BEGIN
   Zulauf_AR_Niv.EW_Peri := 16#287C;
   Zulauf_AR_Niv.EW_PW := 0.0;
   Zulauf_AR_Niv.E.St := FALSE;
   Zulauf_AR_Niv.E.Wt := FALSE;
   Zulauf_AR_Niv.E.Kom_DP := FALSE;
   Zulauf_AR_Niv.E.Kom_int := FALSE;
   Zulauf_AR_Niv.E.int_St := FALSE;
   Zulauf_AR_Niv.E.MW_OF_St := FALSE;
   Zulauf_AR_Niv.E.MW_inv_St := FALSE;
   Zulauf_AR_Niv.E.ZI := FALSE;
   Zulauf_AR_Niv.E.AF_St := FALSE;
   Zulauf_AR_Niv.E.Res09 := FALSE;
   Zulauf_AR_Niv.E.Res10 := FALSE;
   Zulauf_AR_Niv.E.Res11 := FALSE;
   Zulauf_AR_Niv.E.Res12 := FALSE;
   Zulauf_AR_Niv.E.Res13 := FALSE;
   Zulauf_AR_Niv.E.Res14 := FALSE;
   Zulauf_AR_Niv.E.Res15 := FALSE;
   Zulauf_AR_Temp.EW_Peri := 16#1599;
   Zulauf_AR_Temp.EW_PW := 0.0;
   Zulauf_AR_Temp.E.St := FALSE;
   Zulauf_AR_Temp.E.Wt := FALSE;
   Zulauf_AR_Temp.E.Kom_DP := FALSE;
   Zulauf_AR_Temp.E.Kom_int := FALSE;
   Zulauf_AR_Temp.E.int_St := FALSE;
   Zulauf_AR_Temp.E.MW_OF_St := FALSE;
   Zulauf_AR_Temp.E.MW_inv_St := FALSE;
   Zulauf_AR_Temp.E.ZI := FALSE;
   Zulauf_AR_Temp.E.AF_St := FALSE;
   Zulauf_AR_Temp.E.Res09 := FALSE;
   Zulauf_AR_Temp.E.Res10 := FALSE;
   Zulauf_AR_Temp.E.Res11 := FALSE;
   Zulauf_AR_Temp.E.Res12 := FALSE;
   Zulauf_AR_Temp.E.Res13 := FALSE;
   Zulauf_AR_Temp.E.Res14 := FALSE;
   Zulauf_AR_Temp.E.Res15 := FALSE;
   Zulauf_AR_DF.EW_Peri := 16#0000;
   Zulauf_AR_DF.EW_PW := 0.0;
   Zulauf_AR_DF.E.St := FALSE;
   Zulauf_AR_DF.E.Wt := FALSE;
   Zulauf_AR_DF.E.Kom_DP := FALSE;
   Zulauf_AR_DF.E.Kom_int := FALSE;
   Zulauf_AR_DF.E.int_St := FALSE;
   Zulauf_AR_DF.E.MW_OF_St := FALSE;
   Zulauf_AR_DF.E.MW_inv_St := FALSE;
   Zulauf_AR_DF.E.ZI := FALSE;
   Zulauf_AR_DF.E.AF_St := FALSE;
   Zulauf_AR_DF.E.Res09 := FALSE;
   Zulauf_AR_DF.E.Res10 := FALSE;
   Zulauf_AR_DF.E.Res11 := FALSE;
   Zulauf_AR_DF.E.Res12 := FALSE;
   Zulauf_AR_DF.E.Res13 := FALSE;
   Zulauf_AR_DF.E.Res14 := FALSE;
   Zulauf_AR_DF.E.Res15 := FALSE;
   BB1_AS1_SS.EW_Peri := 16#1599;
   BB1_AS1_SS.EW_PW := 0.0;
   BB1_AS1_SS.E.St := FALSE;
   BB1_AS1_SS.E.Wt := FALSE;
   BB1_AS1_SS.E.Kom_DP := FALSE;
   BB1_AS1_SS.E.Kom_int := FALSE;
   BB1_AS1_SS.E.int_St := FALSE;
   BB1_AS1_SS.E.MW_OF_St := FALSE;
   BB1_AS1_SS.E.MW_inv_St := FALSE;
   BB1_AS1_SS.E.ZI := FALSE;
   BB1_AS1_SS.E.AF_St := FALSE;
   BB1_AS1_SS.E.Res09 := FALSE;
   BB1_AS1_SS.E.Res10 := FALSE;
   BB1_AS1_SS.E.Res11 := FALSE;
   BB1_AS1_SS.E.Res12 := FALSE;
   BB1_AS1_SS.E.Res13 := FALSE;
   BB1_AS1_SS.E.Res14 := FALSE;
   BB1_AS1_SS.E.Res15 := FALSE;
   BB1_AS2_SS.EW_Peri := 16#57CD;
   BB1_AS2_SS.EW_PW := 0.0;
   BB1_AS2_SS.E.St := FALSE;
   BB1_AS2_SS.E.Wt := FALSE;
   BB1_AS2_SS.E.Kom_DP := FALSE;
   BB1_AS2_SS.E.Kom_int := FALSE;
   BB1_AS2_SS.E.int_St := FALSE;
   BB1_AS2_SS.E.MW_OF_St := FALSE;
   BB1_AS2_SS.E.MW_inv_St := FALSE;
   BB1_AS2_SS.E.ZI := FALSE;
   BB1_AS2_SS.E.AF_St := FALSE;
   BB1_AS2_SS.E.Res09 := FALSE;
   BB1_AS2_SS.E.Res10 := FALSE;
   BB1_AS2_SS.E.Res11 := FALSE;
   BB1_AS2_SS.E.Res12 := FALSE;
   BB1_AS2_SS.E.Res13 := FALSE;
   BB1_AS2_SS.E.Res14 := FALSE;
   BB1_AS2_SS.E.Res15 := FALSE;
   BB2_AS1_SS.EW_Peri := 16#15A5;
   BB2_AS1_SS.EW_PW := 0.0;
   BB2_AS1_SS.E.St := FALSE;
   BB2_AS1_SS.E.Wt := FALSE;
   BB2_AS1_SS.E.Kom_DP := FALSE;
   BB2_AS1_SS.E.Kom_int := FALSE;
   BB2_AS1_SS.E.int_St := FALSE;
   BB2_AS1_SS.E.MW_OF_St := FALSE;
   BB2_AS1_SS.E.MW_inv_St := FALSE;
   BB2_AS1_SS.E.ZI := FALSE;
   BB2_AS1_SS.E.AF_St := FALSE;
   BB2_AS1_SS.E.Res09 := FALSE;
   BB2_AS1_SS.E.Res10 := FALSE;
   BB2_AS1_SS.E.Res11 := FALSE;
   BB2_AS1_SS.E.Res12 := FALSE;
   BB2_AS1_SS.E.Res13 := FALSE;
   BB2_AS1_SS.E.Res14 := FALSE;
   BB2_AS1_SS.E.Res15 := FALSE;
   BB2_AS2_SS.EW_Peri := 16#15B8;
   BB2_AS2_SS.EW_PW := 0.0;
   BB2_AS2_SS.E.St := FALSE;
   BB2_AS2_SS.E.Wt := FALSE;
   BB2_AS2_SS.E.Kom_DP := FALSE;
   BB2_AS2_SS.E.Kom_int := FALSE;
   BB2_AS2_SS.E.int_St := FALSE;
   BB2_AS2_SS.E.MW_OF_St := FALSE;
   BB2_AS2_SS.E.MW_inv_St := FALSE;
   BB2_AS2_SS.E.ZI := FALSE;
   BB2_AS2_SS.E.AF_St := FALSE;
   BB2_AS2_SS.E.Res09 := FALSE;
   BB2_AS2_SS.E.Res10 := FALSE;
   BB2_AS2_SS.E.Res11 := FALSE;
   BB2_AS2_SS.E.Res12 := FALSE;
   BB2_AS2_SS.E.Res13 := FALSE;
   BB2_AS2_SS.E.Res14 := FALSE;
   BB2_AS2_SS.E.Res15 := FALSE;
   BB1_O2.EW_Peri := 16#235C;
   BB1_O2.EW_PW := 0.0;
   BB1_O2.E.St := FALSE;
   BB1_O2.E.Wt := FALSE;
   BB1_O2.E.Kom_DP := FALSE;
   BB1_O2.E.Kom_int := FALSE;
   BB1_O2.E.int_St := FALSE;
   BB1_O2.E.MW_OF_St := FALSE;
   BB1_O2.E.MW_inv_St := FALSE;
   BB1_O2.E.ZI := FALSE;
   BB1_O2.E.AF_St := FALSE;
   BB1_O2.E.Res09 := FALSE;
   BB1_O2.E.Res10 := FALSE;
   BB1_O2.E.Res11 := FALSE;
   BB1_O2.E.Res12 := FALSE;
   BB1_O2.E.Res13 := FALSE;
   BB1_O2.E.Res14 := FALSE;
   BB1_O2.E.Res15 := FALSE;
   BB1_Temp.EW_Peri := 16#2EBA;
   BB1_Temp.EW_PW := 0.0;
   BB1_Temp.E.St := FALSE;
   BB1_Temp.E.Wt := FALSE;
   BB1_Temp.E.Kom_DP := FALSE;
   BB1_Temp.E.Kom_int := FALSE;
   BB1_Temp.E.int_St := FALSE;
   BB1_Temp.E.MW_OF_St := FALSE;
   BB1_Temp.E.MW_inv_St := FALSE;
   BB1_Temp.E.ZI := FALSE;
   BB1_Temp.E.AF_St := FALSE;
   BB1_Temp.E.Res09 := FALSE;
   BB1_Temp.E.Res10 := FALSE;
   BB1_Temp.E.Res11 := FALSE;
   BB1_Temp.E.Res12 := FALSE;
   BB1_Temp.E.Res13 := FALSE;
   BB1_Temp.E.Res14 := FALSE;
   BB1_Temp.E.Res15 := FALSE;
   BB2_O2.EW_Peri := 16#2288;
   BB2_O2.EW_PW := 0.0;
   BB2_O2.E.St := FALSE;
   BB2_O2.E.Wt := FALSE;
   BB2_O2.E.Kom_DP := FALSE;
   BB2_O2.E.Kom_int := FALSE;
   BB2_O2.E.int_St := FALSE;
   BB2_O2.E.MW_OF_St := FALSE;
   BB2_O2.E.MW_inv_St := FALSE;
   BB2_O2.E.ZI := FALSE;
   BB2_O2.E.AF_St := FALSE;
   BB2_O2.E.Res09 := FALSE;
   BB2_O2.E.Res10 := FALSE;
   BB2_O2.E.Res11 := FALSE;
   BB2_O2.E.Res12 := FALSE;
   BB2_O2.E.Res13 := FALSE;
   BB2_O2.E.Res14 := FALSE;
   BB2_O2.E.Res15 := FALSE;
   BB2_Temp.EW_Peri := 16#2E74;
   BB2_Temp.EW_PW := 0.0;
   BB2_Temp.E.St := FALSE;
   BB2_Temp.E.Wt := FALSE;
   BB2_Temp.E.Kom_DP := FALSE;
   BB2_Temp.E.Kom_int := FALSE;
   BB2_Temp.E.int_St := FALSE;
   BB2_Temp.E.MW_OF_St := FALSE;
   BB2_Temp.E.MW_inv_St := FALSE;
   BB2_Temp.E.ZI := FALSE;
   BB2_Temp.E.AF_St := FALSE;
   BB2_Temp.E.Res09 := FALSE;
   BB2_Temp.E.Res10 := FALSE;
   BB2_Temp.E.Res11 := FALSE;
   BB2_Temp.E.Res12 := FALSE;
   BB2_Temp.E.Res13 := FALSE;
   BB2_Temp.E.Res14 := FALSE;
   BB2_Temp.E.Res15 := FALSE;
   BB1_DF.EW_Peri := 16#1599;
   BB1_DF.EW_PW := 0.0;
   BB1_DF.E.St := FALSE;
   BB1_DF.E.Wt := FALSE;
   BB1_DF.E.Kom_DP := FALSE;
   BB1_DF.E.Kom_int := FALSE;
   BB1_DF.E.int_St := FALSE;
   BB1_DF.E.MW_OF_St := FALSE;
   BB1_DF.E.MW_inv_St := FALSE;
   BB1_DF.E.ZI := FALSE;
   BB1_DF.E.AF_St := FALSE;
   BB1_DF.E.Res09 := FALSE;
   BB1_DF.E.Res10 := FALSE;
   BB1_DF.E.Res11 := FALSE;
   BB1_DF.E.Res12 := FALSE;
   BB1_DF.E.Res13 := FALSE;
   BB1_DF.E.Res14 := FALSE;
   BB1_DF.E.Res15 := FALSE;
   BB2_DF.EW_Peri := 16#1599;
   BB2_DF.EW_PW := 0.0;
   BB2_DF.E.St := FALSE;
   BB2_DF.E.Wt := FALSE;
   BB2_DF.E.Kom_DP := FALSE;
   BB2_DF.E.Kom_int := FALSE;
   BB2_DF.E.int_St := FALSE;
   BB2_DF.E.MW_OF_St := FALSE;
   BB2_DF.E.MW_inv_St := FALSE;
   BB2_DF.E.ZI := FALSE;
   BB2_DF.E.AF_St := FALSE;
   BB2_DF.E.Res09 := FALSE;
   BB2_DF.E.Res10 := FALSE;
   BB2_DF.E.Res11 := FALSE;
   BB2_DF.E.Res12 := FALSE;
   BB2_DF.E.Res13 := FALSE;
   BB2_DF.E.Res14 := FALSE;
   BB2_DF.E.Res15 := FALSE;
   Zulauf_Niv.EW_Peri := 16#2C3F;
   Zulauf_Niv.EW_PW := 0.0;
   Zulauf_Niv.E.St := FALSE;
   Zulauf_Niv.E.Wt := FALSE;
   Zulauf_Niv.E.Kom_DP := FALSE;
   Zulauf_Niv.E.Kom_int := FALSE;
   Zulauf_Niv.E.int_St := FALSE;
   Zulauf_Niv.E.MW_OF_St := FALSE;
   Zulauf_Niv.E.MW_inv_St := FALSE;
   Zulauf_Niv.E.ZI := FALSE;
   Zulauf_Niv.E.AF_St := FALSE;
   Zulauf_Niv.E.Res09 := FALSE;
   Zulauf_Niv.E.Res10 := FALSE;
   Zulauf_Niv.E.Res11 := FALSE;
   Zulauf_Niv.E.Res12 := FALSE;
   Zulauf_Niv.E.Res13 := FALSE;
   Zulauf_Niv.E.Res14 := FALSE;
   Zulauf_Niv.E.Res15 := FALSE;
   Zulauf_DF.EW_Peri := 16#39D4;
   Zulauf_DF.EW_PW := 0.0;
   Zulauf_DF.E.St := FALSE;
   Zulauf_DF.E.Wt := FALSE;
   Zulauf_DF.E.Kom_DP := FALSE;
   Zulauf_DF.E.Kom_int := FALSE;
   Zulauf_DF.E.int_St := FALSE;
   Zulauf_DF.E.MW_OF_St := FALSE;
   Zulauf_DF.E.MW_inv_St := FALSE;
   Zulauf_DF.E.ZI := FALSE;
   Zulauf_DF.E.AF_St := FALSE;
   Zulauf_DF.E.Res09 := FALSE;
   Zulauf_DF.E.Res10 := FALSE;
   Zulauf_DF.E.Res11 := FALSE;
   Zulauf_DF.E.Res12 := FALSE;
   Zulauf_DF.E.Res13 := FALSE;
   Zulauf_DF.E.Res14 := FALSE;
   Zulauf_DF.E.Res15 := FALSE;
   Verteiler_pH.EW_Peri := 16#1599;
   Verteiler_pH.EW_PW := 0.0;
   Verteiler_pH.E.St := FALSE;
   Verteiler_pH.E.Wt := FALSE;
   Verteiler_pH.E.Kom_DP := FALSE;
   Verteiler_pH.E.Kom_int := FALSE;
   Verteiler_pH.E.int_St := FALSE;
   Verteiler_pH.E.MW_OF_St := FALSE;
   Verteiler_pH.E.MW_inv_St := FALSE;
   Verteiler_pH.E.ZI := FALSE;
   Verteiler_pH.E.AF_St := FALSE;
   Verteiler_pH.E.Res09 := FALSE;
   Verteiler_pH.E.Res10 := FALSE;
   Verteiler_pH.E.Res11 := FALSE;
   Verteiler_pH.E.Res12 := FALSE;
   Verteiler_pH.E.Res13 := FALSE;
   Verteiler_pH.E.Res14 := FALSE;
   Verteiler_pH.E.Res15 := FALSE;
   Verteiler_O2.EW_Peri := 16#1599;
   Verteiler_O2.EW_PW := 0.0;
   Verteiler_O2.E.St := FALSE;
   Verteiler_O2.E.Wt := FALSE;
   Verteiler_O2.E.Kom_DP := FALSE;
   Verteiler_O2.E.Kom_int := FALSE;
   Verteiler_O2.E.int_St := FALSE;
   Verteiler_O2.E.MW_OF_St := FALSE;
   Verteiler_O2.E.MW_inv_St := FALSE;
   Verteiler_O2.E.ZI := FALSE;
   Verteiler_O2.E.AF_St := FALSE;
   Verteiler_O2.E.Res09 := FALSE;
   Verteiler_O2.E.Res10 := FALSE;
   Verteiler_O2.E.Res11 := FALSE;
   Verteiler_O2.E.Res12 := FALSE;
   Verteiler_O2.E.Res13 := FALSE;
   Verteiler_O2.E.Res14 := FALSE;
   Verteiler_O2.E.Res15 := FALSE;
   Verteiler_Temp.EW_Peri := 16#1599;
   Verteiler_Temp.EW_PW := 0.0;
   Verteiler_Temp.E.St := FALSE;
   Verteiler_Temp.E.Wt := FALSE;
   Verteiler_Temp.E.Kom_DP := FALSE;
   Verteiler_Temp.E.Kom_int := FALSE;
   Verteiler_Temp.E.int_St := FALSE;
   Verteiler_Temp.E.MW_OF_St := FALSE;
   Verteiler_Temp.E.MW_inv_St := FALSE;
   Verteiler_Temp.E.ZI := FALSE;
   Verteiler_Temp.E.AF_St := FALSE;
   Verteiler_Temp.E.Res09 := FALSE;
   Verteiler_Temp.E.Res10 := FALSE;
   Verteiler_Temp.E.Res11 := FALSE;
   Verteiler_Temp.E.Res12 := FALSE;
   Verteiler_Temp.E.Res13 := FALSE;
   Verteiler_Temp.E.Res14 := FALSE;
   Verteiler_Temp.E.Res15 := FALSE;
   BB_UeSS_DF.EW_Peri := 16#1592;
   BB_UeSS_DF.EW_PW := 0.0;
   BB_UeSS_DF.E.St := FALSE;
   BB_UeSS_DF.E.Wt := FALSE;
   BB_UeSS_DF.E.Kom_DP := FALSE;
   BB_UeSS_DF.E.Kom_int := FALSE;
   BB_UeSS_DF.E.int_St := FALSE;
   BB_UeSS_DF.E.MW_OF_St := FALSE;
   BB_UeSS_DF.E.MW_inv_St := FALSE;
   BB_UeSS_DF.E.ZI := FALSE;
   BB_UeSS_DF.E.AF_St := FALSE;
   BB_UeSS_DF.E.Res09 := FALSE;
   BB_UeSS_DF.E.Res10 := FALSE;
   BB_UeSS_DF.E.Res11 := FALSE;
   BB_UeSS_DF.E.Res12 := FALSE;
   BB_UeSS_DF.E.Res13 := FALSE;
   BB_UeSS_DF.E.Res14 := FALSE;
   BB_UeSS_DF.E.Res15 := FALSE;
   Ablauf_DF.EW_Peri := 16#35E9;
   Ablauf_DF.EW_PW := 0.0;
   Ablauf_DF.E.St := FALSE;
   Ablauf_DF.E.Wt := FALSE;
   Ablauf_DF.E.Kom_DP := FALSE;
   Ablauf_DF.E.Kom_int := FALSE;
   Ablauf_DF.E.int_St := FALSE;
   Ablauf_DF.E.MW_OF_St := FALSE;
   Ablauf_DF.E.MW_inv_St := FALSE;
   Ablauf_DF.E.ZI := FALSE;
   Ablauf_DF.E.AF_St := FALSE;
   Ablauf_DF.E.Res09 := FALSE;
   Ablauf_DF.E.Res10 := FALSE;
   Ablauf_DF.E.Res11 := FALSE;
   Ablauf_DF.E.Res12 := FALSE;
   Ablauf_DF.E.Res13 := FALSE;
   Ablauf_DF.E.Res14 := FALSE;
   Ablauf_DF.E.Res15 := FALSE;
   Ablauf_pH.EW_Peri := 16#4122;
   Ablauf_pH.EW_PW := 0.0;
   Ablauf_pH.E.St := FALSE;
   Ablauf_pH.E.Wt := FALSE;
   Ablauf_pH.E.Kom_DP := FALSE;
   Ablauf_pH.E.Kom_int := FALSE;
   Ablauf_pH.E.int_St := FALSE;
   Ablauf_pH.E.MW_OF_St := FALSE;
   Ablauf_pH.E.MW_inv_St := FALSE;
   Ablauf_pH.E.ZI := FALSE;
   Ablauf_pH.E.AF_St := FALSE;
   Ablauf_pH.E.Res09 := FALSE;
   Ablauf_pH.E.Res10 := FALSE;
   Ablauf_pH.E.Res11 := FALSE;
   Ablauf_pH.E.Res12 := FALSE;
   Ablauf_pH.E.Res13 := FALSE;
   Ablauf_pH.E.Res14 := FALSE;
   Ablauf_pH.E.Res15 := FALSE;
   Ablauf_O2.EW_Peri := 16#225E;
   Ablauf_O2.EW_PW := 0.0;
   Ablauf_O2.E.St := FALSE;
   Ablauf_O2.E.Wt := FALSE;
   Ablauf_O2.E.Kom_DP := FALSE;
   Ablauf_O2.E.Kom_int := FALSE;
   Ablauf_O2.E.int_St := FALSE;
   Ablauf_O2.E.MW_OF_St := FALSE;
   Ablauf_O2.E.MW_inv_St := FALSE;
   Ablauf_O2.E.ZI := FALSE;
   Ablauf_O2.E.AF_St := FALSE;
   Ablauf_O2.E.Res09 := FALSE;
   Ablauf_O2.E.Res10 := FALSE;
   Ablauf_O2.E.Res11 := FALSE;
   Ablauf_O2.E.Res12 := FALSE;
   Ablauf_O2.E.Res13 := FALSE;
   Ablauf_O2.E.Res14 := FALSE;
   Ablauf_O2.E.Res15 := FALSE;
   Ablauf_Temp.EW_Peri := 16#2BEC;
   Ablauf_Temp.EW_PW := 0.0;
   Ablauf_Temp.E.St := FALSE;
   Ablauf_Temp.E.Wt := FALSE;
   Ablauf_Temp.E.Kom_DP := FALSE;
   Ablauf_Temp.E.Kom_int := FALSE;
   Ablauf_Temp.E.int_St := FALSE;
   Ablauf_Temp.E.MW_OF_St := FALSE;
   Ablauf_Temp.E.MW_inv_St := FALSE;
   Ablauf_Temp.E.ZI := FALSE;
   Ablauf_Temp.E.AF_St := FALSE;
   Ablauf_Temp.E.Res09 := FALSE;
   Ablauf_Temp.E.Res10 := FALSE;
   Ablauf_Temp.E.Res11 := FALSE;
   Ablauf_Temp.E.Res12 := FALSE;
   Ablauf_Temp.E.Res13 := FALSE;
   Ablauf_Temp.E.Res14 := FALSE;
   Ablauf_Temp.E.Res15 := FALSE;
   Schlamm_ED_Niv.EW_Peri := 16#1599;
   Schlamm_ED_Niv.EW_PW := 0.0;
   Schlamm_ED_Niv.E.St := FALSE;
   Schlamm_ED_Niv.E.Wt := FALSE;
   Schlamm_ED_Niv.E.Kom_DP := FALSE;
   Schlamm_ED_Niv.E.Kom_int := FALSE;
   Schlamm_ED_Niv.E.int_St := FALSE;
   Schlamm_ED_Niv.E.MW_OF_St := FALSE;
   Schlamm_ED_Niv.E.MW_inv_St := FALSE;
   Schlamm_ED_Niv.E.ZI := FALSE;
   Schlamm_ED_Niv.E.AF_St := FALSE;
   Schlamm_ED_Niv.E.Res09 := FALSE;
   Schlamm_ED_Niv.E.Res10 := FALSE;
   Schlamm_ED_Niv.E.Res11 := FALSE;
   Schlamm_ED_Niv.E.Res12 := FALSE;
   Schlamm_ED_Niv.E.Res13 := FALSE;
   Schlamm_ED_Niv.E.Res14 := FALSE;
   Schlamm_ED_Niv.E.Res15 := FALSE;
   Schlamm_Besch_Niv.EW_Peri := 16#1599;
   Schlamm_Besch_Niv.EW_PW := 0.0;
   Schlamm_Besch_Niv.E.St := FALSE;
   Schlamm_Besch_Niv.E.Wt := FALSE;
   Schlamm_Besch_Niv.E.Kom_DP := FALSE;
   Schlamm_Besch_Niv.E.Kom_int := FALSE;
   Schlamm_Besch_Niv.E.int_St := FALSE;
   Schlamm_Besch_Niv.E.MW_OF_St := FALSE;
   Schlamm_Besch_Niv.E.MW_inv_St := FALSE;
   Schlamm_Besch_Niv.E.ZI := FALSE;
   Schlamm_Besch_Niv.E.AF_St := FALSE;
   Schlamm_Besch_Niv.E.Res09 := FALSE;
   Schlamm_Besch_Niv.E.Res10 := FALSE;
   Schlamm_Besch_Niv.E.Res11 := FALSE;
   Schlamm_Besch_Niv.E.Res12 := FALSE;
   Schlamm_Besch_Niv.E.Res13 := FALSE;
   Schlamm_Besch_Niv.E.Res14 := FALSE;
   Schlamm_Besch_Niv.E.Res15 := FALSE;
   Schlamm_Besch_DF.EW_Peri := 16#159B;
   Schlamm_Besch_DF.EW_PW := 0.0;
   Schlamm_Besch_DF.E.St := FALSE;
   Schlamm_Besch_DF.E.Wt := FALSE;
   Schlamm_Besch_DF.E.Kom_DP := FALSE;
   Schlamm_Besch_DF.E.Kom_int := FALSE;
   Schlamm_Besch_DF.E.int_St := FALSE;
   Schlamm_Besch_DF.E.MW_OF_St := FALSE;
   Schlamm_Besch_DF.E.MW_inv_St := FALSE;
   Schlamm_Besch_DF.E.ZI := FALSE;
   Schlamm_Besch_DF.E.AF_St := FALSE;
   Schlamm_Besch_DF.E.Res09 := FALSE;
   Schlamm_Besch_DF.E.Res10 := FALSE;
   Schlamm_Besch_DF.E.Res11 := FALSE;
   Schlamm_Besch_DF.E.Res12 := FALSE;
   Schlamm_Besch_DF.E.Res13 := FALSE;
   Schlamm_Besch_DF.E.Res14 := FALSE;
   Schlamm_Besch_DF.E.Res15 := FALSE;
   Truebwasser_Niv.EW_Peri := 16#28E3;
   Truebwasser_Niv.EW_PW := 0.0;
   Truebwasser_Niv.E.St := FALSE;
   Truebwasser_Niv.E.Wt := FALSE;
   Truebwasser_Niv.E.Kom_DP := FALSE;
   Truebwasser_Niv.E.Kom_int := FALSE;
   Truebwasser_Niv.E.int_St := FALSE;
   Truebwasser_Niv.E.MW_OF_St := FALSE;
   Truebwasser_Niv.E.MW_inv_St := FALSE;
   Truebwasser_Niv.E.ZI := FALSE;
   Truebwasser_Niv.E.AF_St := FALSE;
   Truebwasser_Niv.E.Res09 := FALSE;
   Truebwasser_Niv.E.Res10 := FALSE;
   Truebwasser_Niv.E.Res11 := FALSE;
   Truebwasser_Niv.E.Res12 := FALSE;
   Truebwasser_Niv.E.Res13 := FALSE;
   Truebwasser_Niv.E.Res14 := FALSE;
   Truebwasser_Niv.E.Res15 := FALSE;
   Truebwasser_DF.EW_Peri := 16#1597;
   Truebwasser_DF.EW_PW := 0.0;
   Truebwasser_DF.E.St := FALSE;
   Truebwasser_DF.E.Wt := FALSE;
   Truebwasser_DF.E.Kom_DP := FALSE;
   Truebwasser_DF.E.Kom_int := FALSE;
   Truebwasser_DF.E.int_St := FALSE;
   Truebwasser_DF.E.MW_OF_St := FALSE;
   Truebwasser_DF.E.MW_inv_St := FALSE;
   Truebwasser_DF.E.ZI := FALSE;
   Truebwasser_DF.E.AF_St := FALSE;
   Truebwasser_DF.E.Res09 := FALSE;
   Truebwasser_DF.E.Res10 := FALSE;
   Truebwasser_DF.E.Res11 := FALSE;
   Truebwasser_DF.E.Res12 := FALSE;
   Truebwasser_DF.E.Res13 := FALSE;
   Truebwasser_DF.E.Res14 := FALSE;
   Truebwasser_DF.E.Res15 := FALSE;
   Zulauf_SF_Niv.EW_Peri := 16#1599;
   Zulauf_SF_Niv.EW_PW := 0.0;
   Zulauf_SF_Niv.E.St := FALSE;
   Zulauf_SF_Niv.E.Wt := FALSE;
   Zulauf_SF_Niv.E.Kom_DP := FALSE;
   Zulauf_SF_Niv.E.Kom_int := FALSE;
   Zulauf_SF_Niv.E.int_St := FALSE;
   Zulauf_SF_Niv.E.MW_OF_St := FALSE;
   Zulauf_SF_Niv.E.MW_inv_St := FALSE;
   Zulauf_SF_Niv.E.ZI := FALSE;
   Zulauf_SF_Niv.E.AF_St := FALSE;
   Zulauf_SF_Niv.E.Res09 := FALSE;
   Zulauf_SF_Niv.E.Res10 := FALSE;
   Zulauf_SF_Niv.E.Res11 := FALSE;
   Zulauf_SF_Niv.E.Res12 := FALSE;
   Zulauf_SF_Niv.E.Res13 := FALSE;
   Zulauf_SF_Niv.E.Res14 := FALSE;
   Zulauf_SF_Niv.E.Res15 := FALSE;
   Ablauf_NOx.EW_Peri := 16#1BEB;
   Ablauf_NOx.EW_PW := 0.0;
   Ablauf_NOx.E.St := FALSE;
   Ablauf_NOx.E.Wt := FALSE;
   Ablauf_NOx.E.Kom_DP := FALSE;
   Ablauf_NOx.E.Kom_int := FALSE;
   Ablauf_NOx.E.int_St := FALSE;
   Ablauf_NOx.E.MW_OF_St := FALSE;
   Ablauf_NOx.E.MW_inv_St := FALSE;
   Ablauf_NOx.E.ZI := FALSE;
   Ablauf_NOx.E.AF_St := FALSE;
   Ablauf_NOx.E.Res09 := FALSE;
   Ablauf_NOx.E.Res10 := FALSE;
   Ablauf_NOx.E.Res11 := FALSE;
   Ablauf_NOx.E.Res12 := FALSE;
   Ablauf_NOx.E.Res13 := FALSE;
   Ablauf_NOx.E.Res14 := FALSE;
   Ablauf_NOx.E.Res15 := FALSE;
   Ablauf_PO4.EW_Peri := 16#218F;
   Ablauf_PO4.EW_PW := 0.0;
   Ablauf_PO4.E.St := FALSE;
   Ablauf_PO4.E.Wt := FALSE;
   Ablauf_PO4.E.Kom_DP := FALSE;
   Ablauf_PO4.E.Kom_int := FALSE;
   Ablauf_PO4.E.int_St := FALSE;
   Ablauf_PO4.E.MW_OF_St := FALSE;
   Ablauf_PO4.E.MW_inv_St := FALSE;
   Ablauf_PO4.E.ZI := FALSE;
   Ablauf_PO4.E.AF_St := FALSE;
   Ablauf_PO4.E.Res09 := FALSE;
   Ablauf_PO4.E.Res10 := FALSE;
   Ablauf_PO4.E.Res11 := FALSE;
   Ablauf_PO4.E.Res12 := FALSE;
   Ablauf_PO4.E.Res13 := FALSE;
   Ablauf_PO4.E.Res14 := FALSE;
   Ablauf_PO4.E.Res15 := FALSE;

END_DATA_BLOCK

DATA_BLOCK "DB118_PW_Meld"
{ S7_Optimized_Access := 'FALSE' }
VERSION : 0.1
NON_RETAIN
   STRUCT
      FW_APW_Oeb_KB { S7_SetPoint := 'False'} : "T_PW_MELD";   // Oebisfelde APW Krumme Breite
      FW_APW_BrR_DM : "T_PW_MELD";   // Breitenrode APW Denkmal
      FW_APW_Oeb_Tu : "T_PW_MELD";   // Oebisfelde APW Tunnel
      FW_APW_Oeb_KS : "T_PW_MELD";   // Oebisfelde APW Klötzer Str.
      FW_APW_Oeb_PG : "T_PW_MELD";   // Oebisfelde APW Papengraben
      FW_APW_Oeb_LW : "T_PW_MELD";   // Oebisfelde APW Lehmweg
      FW_APW_GeD_WG : "T_PW_MELD";   // Gehrendorf APW Wiesengrund
      FW_APW_GeD_AA : "T_PW_MELD";   // Gehrendorf APW An der Aller
      FW_APW_WaD : "T_PW_MELD";   // Wassensdorf APW
      FW_APW_WeD : "T_PW_MELD";   // Weddendorf APW
      FW_APW_NiD : "T_PW_MELD";   // Niendorf APW
      FW_APW_LoS : "T_PW_MELD";   // Lockstedt APW
      FW_APW_Oeb_Ge : "T_PW_MELD";   // Oebisfelde APW Gewerbe
      FW_APW_BuH : "T_PW_MELD";   // Buchhorst APW
      FW_APW_BrR_TS : "T_PW_MELD";   // Breitenrode APW Trafostation
   END_STRUCT;


BEGIN

END_DATA_BLOCK

DATA_BLOCK "DB119_PW_Bef"
{ S7_Optimized_Access := 'FALSE' }
VERSION : 0.1
NON_RETAIN
   STRUCT
      FW_APW_Oeb_KB { S7_SetPoint := 'False'} : "T_PW_BEF";   // Oebisfelde APW Krumme Breite
      FW_APW_BrR_DM : "T_PW_BEF";   // Breitenrode APW Denkmal
      FW_APW_Oeb_Tu : "T_PW_BEF";   // Oebisfelde APW Tunnel
      FW_APW_Oeb_KS : "T_PW_BEF";   // Oebisfelde APW Klötzer Str.
      FW_APW_Oeb_PG : "T_PW_BEF";   // Oebisfelde APW Papengraben
      FW_APW_Oeb_LW : "T_PW_BEF";   // Oebisfelde APW Lehmweg
      FW_APW_GeD_WG : "T_PW_BEF";   // Gehrendorf APW Wiesengrund
      FW_APW_GeD_AA : "T_PW_BEF";   // Gehrendorf APW An der Aller
      FW_APW_WaD : "T_PW_BEF";   // Wassensdorf APW
      FW_APW_WeD : "T_PW_BEF";   // Weddendorf APW
      FW_APW_NiD : "T_PW_BEF";   // Niendorf APW
      FW_APW_LoS : "T_PW_BEF";   // Lockstedt APW
      FW_APW_Oeb_Ge : "T_PW_BEF";   // Oebisfelde APW Gewerbe
      FW_APW_BuH : "T_PW_BEF";   // Buchhorst APW
      FW_APW_BrR_TS : "T_PW_BEF";   // Breitenrode APW Trafostation
   END_STRUCT;


BEGIN

END_DATA_BLOCK

DATA_BLOCK "IDB_FB51_Time"
{ S7_Optimized_Access := 'TRUE' }
VERSION : 0.1
NON_RETAIN
"FB51_Time"

BEGIN
   tm_Array_last[0] := 16#07;
   tm_Array_last[1] := 16#E2;
   tm_Array_last[2] := 16#07;
   tm_Array_last[3] := 16#12;
   tm_Array_last[4] := 16#04;
   tm_Array_last[5] := 16#09;
   tm_Array_last[6] := 16#2D;
   tm_Array_last[7] := 16#01;
   tm_Array_last[8] := 16#38;
   tm_Array_last[9] := 16#9E;
   tm_Array_last[10] := 16#26;
   tm_Array_last[11] := 16#60;
   tm_Array_last[12] := 16#00;

END_DATA_BLOCK

DATA_BLOCK "DB94_AntrStat_chg"
{ S7_Optimized_Access := 'FALSE' }
VERSION : 0.1
NON_RETAIN
   STRUCT
      Status_last : Array[1..144] of DWord;
      UV_Bef_UV_Chg : Array[1..144] of Bool;
      UV_Bef_NHV_Chg : Array[1..144] of Bool;
      UV_Meld_Chg : Array[1..144] of Bool;
      UV_Prm_Chg : Array[1..144] of Bool;
   END_STRUCT;


BEGIN
   Status_last[1] := 16#2841_2020;
   Status_last[2] := 16#1101_2050;
   Status_last[3] := 16#1101_2050;
   Status_last[4] := 16#1101_2052;
   Status_last[5] := 16#2801_2040;
   Status_last[6] := 16#2801_2040;
   Status_last[7] := 16#6800_2421;
   Status_last[8] := 16#6800_2421;
   Status_last[9] := 16#2801_51C1;
   Status_last[10] := 16#6800_2421;
   Status_last[11] := 16#2801_96C2;
   Status_last[12] := 16#2801_92C2;
   Status_last[13] := 16#2801_92C2;
   Status_last[14] := 16#2801_96C2;
   Status_last[15] := 16#6800_2421;
   Status_last[16] := 16#6800_2421;
   Status_last[17] := 16#6800_2421;
   Status_last[18] := 16#2801_92C2;
   Status_last[19] := 16#A800_2822;
   Status_last[20] := 16#A800_2822;
   Status_last[21] := 16#2801_2020;
   Status_last[22] := 16#1801_2041;
   Status_last[23] := 16#0000_0000;
   Status_last[24] := 16#0000_0000;
   Status_last[25] := 16#0000_0000;
   Status_last[26] := 16#0000_0000;
   Status_last[27] := 16#0000_0000;
   Status_last[28] := 16#0000_0000;
   Status_last[29] := 16#0000_0000;
   Status_last[30] := 16#0000_0000;
   Status_last[31] := 16#0000_0000;
   Status_last[32] := 16#0000_0000;
   Status_last[33] := 16#0000_0000;
   Status_last[34] := 16#0000_0000;
   Status_last[35] := 16#0000_0000;
   Status_last[36] := 16#0000_0000;
   Status_last[37] := 16#0000_0000;
   Status_last[38] := 16#0000_0000;
   Status_last[39] := 16#0000_0000;
   Status_last[40] := 16#0000_0000;
   Status_last[41] := 16#0000_0000;
   Status_last[42] := 16#0000_0000;
   Status_last[43] := 16#0000_0000;
   Status_last[44] := 16#0000_0000;
   Status_last[45] := 16#0000_0000;
   Status_last[46] := 16#0000_0000;
   Status_last[47] := 16#0000_0000;
   Status_last[48] := 16#0000_0000;
   Status_last[49] := 16#0000_0000;
   Status_last[50] := 16#0000_0000;
   Status_last[51] := 16#0000_0000;
   Status_last[52] := 16#0000_0000;
   Status_last[53] := 16#0000_0000;
   Status_last[54] := 16#0000_0000;
   Status_last[55] := 16#0000_0000;
   Status_last[56] := 16#0000_0000;
   Status_last[57] := 16#0000_0000;
   Status_last[58] := 16#0000_0000;
   Status_last[59] := 16#0000_0000;
   Status_last[60] := 16#0000_0000;
   Status_last[61] := 16#0000_0000;
   Status_last[62] := 16#0000_0000;
   Status_last[63] := 16#0000_0000;
   Status_last[64] := 16#0000_0000;
   Status_last[65] := 16#0000_0000;
   Status_last[66] := 16#0000_0000;
   Status_last[67] := 16#0000_0000;
   Status_last[68] := 16#0000_0000;
   Status_last[69] := 16#0000_0000;
   Status_last[70] := 16#0000_0000;
   Status_last[71] := 16#0000_0000;
   Status_last[72] := 16#0000_0000;
   Status_last[73] := 16#0000_0000;
   Status_last[74] := 16#0000_0000;
   Status_last[75] := 16#0000_0000;
   Status_last[76] := 16#0000_0000;
   Status_last[77] := 16#0000_0000;
   Status_last[78] := 16#0000_0000;
   Status_last[79] := 16#0000_0000;
   Status_last[80] := 16#0000_0000;
   Status_last[81] := 16#0000_0000;
   Status_last[82] := 16#0000_0000;
   Status_last[83] := 16#0000_0000;
   Status_last[84] := 16#0000_0000;
   Status_last[85] := 16#0000_0000;
   Status_last[86] := 16#0000_0000;
   Status_last[87] := 16#0000_0000;
   Status_last[88] := 16#0000_0000;
   Status_last[89] := 16#0000_0000;
   Status_last[90] := 16#0000_0000;
   Status_last[91] := 16#0000_0000;
   Status_last[92] := 16#0000_0000;
   Status_last[93] := 16#0000_0000;
   Status_last[94] := 16#2801_2020;
   Status_last[95] := 16#2801_2020;
   Status_last[96] := 16#2801_2020;
   Status_last[97] := 16#2841_2020;
   Status_last[98] := 16#2801_2020;
   Status_last[99] := 16#1801_2000;
   Status_last[100] := 16#1801_2800;
   Status_last[101] := 16#A800_2822;
   Status_last[102] := 16#A800_2822;
   Status_last[103] := 16#A800_2822;
   Status_last[104] := 16#A800_2822;
   Status_last[105] := 16#A800_2822;
   Status_last[106] := 16#1801_2000;
   Status_last[107] := 16#1801_2000;
   Status_last[108] := 16#1801_2000;
   Status_last[109] := 16#1801_2000;
   Status_last[110] := 16#1801_2000;
   Status_last[111] := 16#2801_2820;
   Status_last[112] := 16#2801_2820;
   Status_last[113] := 16#2801_2820;
   Status_last[114] := 16#2801_2820;
   Status_last[115] := 16#2801_2020;
   Status_last[116] := 16#2801_2820;
   Status_last[117] := 16#2841_2020;
   Status_last[118] := 16#2801_2020;
   Status_last[119] := 16#2801_2020;
   Status_last[120] := 16#0000_0000;
   Status_last[121] := 16#0000_0000;
   Status_last[122] := 16#0000_0000;
   Status_last[123] := 16#0000_0000;
   Status_last[124] := 16#0000_0000;
   Status_last[125] := 16#0000_0000;
   Status_last[126] := 16#0000_0000;
   Status_last[127] := 16#A800_2822;
   Status_last[128] := 16#A800_2822;
   Status_last[129] := 16#A800_2822;
   Status_last[130] := 16#2801_2020;
   Status_last[131] := 16#2801_2020;
   Status_last[132] := 16#0000_0000;
   Status_last[133] := 16#0000_0000;
   Status_last[134] := 16#0000_0000;
   Status_last[135] := 16#0000_0000;
   Status_last[136] := 16#0000_0000;
   Status_last[137] := 16#0000_0000;
   Status_last[138] := 16#0000_0000;
   Status_last[139] := 16#0000_0000;
   Status_last[140] := 16#0000_0000;
   Status_last[141] := 16#0000_0000;
   Status_last[142] := 16#0000_0000;
   Status_last[143] := 16#0000_0000;
   Status_last[144] := 16#0000_0000;
   UV_Bef_UV_Chg[1] := FALSE;
   UV_Bef_UV_Chg[2] := FALSE;
   UV_Bef_UV_Chg[3] := FALSE;
   UV_Bef_UV_Chg[4] := FALSE;
   UV_Bef_UV_Chg[5] := FALSE;
   UV_Bef_UV_Chg[6] := FALSE;
   UV_Bef_UV_Chg[7] := FALSE;
   UV_Bef_UV_Chg[8] := FALSE;
   UV_Bef_UV_Chg[9] := FALSE;
   UV_Bef_UV_Chg[10] := FALSE;
   UV_Bef_UV_Chg[11] := FALSE;
   UV_Bef_UV_Chg[12] := FALSE;
   UV_Bef_UV_Chg[13] := FALSE;
   UV_Bef_UV_Chg[14] := FALSE;
   UV_Bef_UV_Chg[15] := FALSE;
   UV_Bef_UV_Chg[16] := FALSE;
   UV_Bef_UV_Chg[17] := FALSE;
   UV_Bef_UV_Chg[18] := FALSE;
   UV_Bef_UV_Chg[19] := FALSE;
   UV_Bef_UV_Chg[20] := FALSE;
   UV_Bef_UV_Chg[21] := FALSE;
   UV_Bef_UV_Chg[22] := FALSE;
   UV_Bef_UV_Chg[23] := FALSE;
   UV_Bef_UV_Chg[24] := FALSE;
   UV_Bef_UV_Chg[25] := FALSE;
   UV_Bef_UV_Chg[26] := FALSE;
   UV_Bef_UV_Chg[27] := FALSE;
   UV_Bef_UV_Chg[28] := FALSE;
   UV_Bef_UV_Chg[29] := FALSE;
   UV_Bef_UV_Chg[30] := FALSE;
   UV_Bef_UV_Chg[31] := FALSE;
   UV_Bef_UV_Chg[32] := FALSE;
   UV_Bef_UV_Chg[33] := FALSE;
   UV_Bef_UV_Chg[34] := FALSE;
   UV_Bef_UV_Chg[35] := FALSE;
   UV_Bef_UV_Chg[36] := FALSE;
   UV_Bef_UV_Chg[37] := FALSE;
   UV_Bef_UV_Chg[38] := FALSE;
   UV_Bef_UV_Chg[39] := FALSE;
   UV_Bef_UV_Chg[40] := FALSE;
   UV_Bef_UV_Chg[41] := FALSE;
   UV_Bef_UV_Chg[42] := FALSE;
   UV_Bef_UV_Chg[43] := FALSE;
   UV_Bef_UV_Chg[44] := FALSE;
   UV_Bef_UV_Chg[45] := FALSE;
   UV_Bef_UV_Chg[46] := FALSE;
   UV_Bef_UV_Chg[47] := FALSE;
   UV_Bef_UV_Chg[48] := FALSE;
   UV_Bef_UV_Chg[49] := FALSE;
   UV_Bef_UV_Chg[50] := FALSE;
   UV_Bef_UV_Chg[51] := FALSE;
   UV_Bef_UV_Chg[52] := FALSE;
   UV_Bef_UV_Chg[53] := FALSE;
   UV_Bef_UV_Chg[54] := FALSE;
   UV_Bef_UV_Chg[55] := FALSE;
   UV_Bef_UV_Chg[56] := FALSE;
   UV_Bef_UV_Chg[57] := FALSE;
   UV_Bef_UV_Chg[58] := FALSE;
   UV_Bef_UV_Chg[59] := FALSE;
   UV_Bef_UV_Chg[60] := FALSE;
   UV_Bef_UV_Chg[61] := FALSE;
   UV_Bef_UV_Chg[62] := FALSE;
   UV_Bef_UV_Chg[63] := FALSE;
   UV_Bef_UV_Chg[64] := FALSE;
   UV_Bef_UV_Chg[65] := FALSE;
   UV_Bef_UV_Chg[66] := FALSE;
   UV_Bef_UV_Chg[67] := FALSE;
   UV_Bef_UV_Chg[68] := FALSE;
   UV_Bef_UV_Chg[69] := FALSE;
   UV_Bef_UV_Chg[70] := FALSE;
   UV_Bef_UV_Chg[71] := FALSE;
   UV_Bef_UV_Chg[72] := FALSE;
   UV_Bef_UV_Chg[73] := FALSE;
   UV_Bef_UV_Chg[74] := FALSE;
   UV_Bef_UV_Chg[75] := FALSE;
   UV_Bef_UV_Chg[76] := FALSE;
   UV_Bef_UV_Chg[77] := FALSE;
   UV_Bef_UV_Chg[78] := FALSE;
   UV_Bef_UV_Chg[79] := FALSE;
   UV_Bef_UV_Chg[80] := FALSE;
   UV_Bef_UV_Chg[81] := FALSE;
   UV_Bef_UV_Chg[82] := FALSE;
   UV_Bef_UV_Chg[83] := FALSE;
   UV_Bef_UV_Chg[84] := FALSE;
   UV_Bef_UV_Chg[85] := FALSE;
   UV_Bef_UV_Chg[86] := FALSE;
   UV_Bef_UV_Chg[87] := FALSE;
   UV_Bef_UV_Chg[88] := FALSE;
   UV_Bef_UV_Chg[89] := FALSE;
   UV_Bef_UV_Chg[90] := FALSE;
   UV_Bef_UV_Chg[91] := FALSE;
   UV_Bef_UV_Chg[92] := FALSE;
   UV_Bef_UV_Chg[93] := FALSE;
   UV_Bef_UV_Chg[94] := FALSE;
   UV_Bef_UV_Chg[95] := FALSE;
   UV_Bef_UV_Chg[96] := FALSE;
   UV_Bef_UV_Chg[97] := FALSE;
   UV_Bef_UV_Chg[98] := FALSE;
   UV_Bef_UV_Chg[99] := FALSE;
   UV_Bef_UV_Chg[100] := FALSE;
   UV_Bef_UV_Chg[101] := FALSE;
   UV_Bef_UV_Chg[102] := FALSE;
   UV_Bef_UV_Chg[103] := FALSE;
   UV_Bef_UV_Chg[104] := FALSE;
   UV_Bef_UV_Chg[105] := FALSE;
   UV_Bef_UV_Chg[106] := FALSE;
   UV_Bef_UV_Chg[107] := FALSE;
   UV_Bef_UV_Chg[108] := FALSE;
   UV_Bef_UV_Chg[109] := FALSE;
   UV_Bef_UV_Chg[110] := FALSE;
   UV_Bef_UV_Chg[111] := FALSE;
   UV_Bef_UV_Chg[112] := FALSE;
   UV_Bef_UV_Chg[113] := FALSE;
   UV_Bef_UV_Chg[114] := FALSE;
   UV_Bef_UV_Chg[115] := FALSE;
   UV_Bef_UV_Chg[116] := FALSE;
   UV_Bef_UV_Chg[117] := FALSE;
   UV_Bef_UV_Chg[118] := FALSE;
   UV_Bef_UV_Chg[119] := FALSE;
   UV_Bef_UV_Chg[120] := FALSE;
   UV_Bef_UV_Chg[121] := FALSE;
   UV_Bef_UV_Chg[122] := FALSE;
   UV_Bef_UV_Chg[123] := FALSE;
   UV_Bef_UV_Chg[124] := FALSE;
   UV_Bef_UV_Chg[125] := FALSE;
   UV_Bef_UV_Chg[126] := FALSE;
   UV_Bef_UV_Chg[127] := FALSE;
   UV_Bef_UV_Chg[128] := FALSE;
   UV_Bef_UV_Chg[129] := FALSE;
   UV_Bef_UV_Chg[130] := FALSE;
   UV_Bef_UV_Chg[131] := FALSE;
   UV_Bef_UV_Chg[132] := FALSE;
   UV_Bef_UV_Chg[133] := FALSE;
   UV_Bef_UV_Chg[134] := FALSE;
   UV_Bef_UV_Chg[135] := FALSE;
   UV_Bef_UV_Chg[136] := FALSE;
   UV_Bef_UV_Chg[137] := FALSE;
   UV_Bef_UV_Chg[138] := FALSE;
   UV_Bef_UV_Chg[139] := FALSE;
   UV_Bef_UV_Chg[140] := FALSE;
   UV_Bef_UV_Chg[141] := FALSE;
   UV_Bef_UV_Chg[142] := FALSE;
   UV_Bef_UV_Chg[143] := FALSE;
   UV_Bef_UV_Chg[144] := FALSE;
   UV_Bef_NHV_Chg[1] := FALSE;
   UV_Bef_NHV_Chg[2] := FALSE;
   UV_Bef_NHV_Chg[3] := FALSE;
   UV_Bef_NHV_Chg[4] := FALSE;
   UV_Bef_NHV_Chg[5] := FALSE;
   UV_Bef_NHV_Chg[6] := FALSE;
   UV_Bef_NHV_Chg[7] := FALSE;
   UV_Bef_NHV_Chg[8] := FALSE;
   UV_Bef_NHV_Chg[9] := FALSE;
   UV_Bef_NHV_Chg[10] := FALSE;
   UV_Bef_NHV_Chg[11] := FALSE;
   UV_Bef_NHV_Chg[12] := FALSE;
   UV_Bef_NHV_Chg[13] := FALSE;
   UV_Bef_NHV_Chg[14] := FALSE;
   UV_Bef_NHV_Chg[15] := FALSE;
   UV_Bef_NHV_Chg[16] := FALSE;
   UV_Bef_NHV_Chg[17] := FALSE;
   UV_Bef_NHV_Chg[18] := FALSE;
   UV_Bef_NHV_Chg[19] := FALSE;
   UV_Bef_NHV_Chg[20] := FALSE;
   UV_Bef_NHV_Chg[21] := FALSE;
   UV_Bef_NHV_Chg[22] := FALSE;
   UV_Bef_NHV_Chg[23] := FALSE;
   UV_Bef_NHV_Chg[24] := FALSE;
   UV_Bef_NHV_Chg[25] := FALSE;
   UV_Bef_NHV_Chg[26] := FALSE;
   UV_Bef_NHV_Chg[27] := FALSE;
   UV_Bef_NHV_Chg[28] := FALSE;
   UV_Bef_NHV_Chg[29] := FALSE;
   UV_Bef_NHV_Chg[30] := FALSE;
   UV_Bef_NHV_Chg[31] := FALSE;
   UV_Bef_NHV_Chg[32] := FALSE;
   UV_Bef_NHV_Chg[33] := FALSE;
   UV_Bef_NHV_Chg[34] := FALSE;
   UV_Bef_NHV_Chg[35] := FALSE;
   UV_Bef_NHV_Chg[36] := FALSE;
   UV_Bef_NHV_Chg[37] := FALSE;
   UV_Bef_NHV_Chg[38] := FALSE;
   UV_Bef_NHV_Chg[39] := FALSE;
   UV_Bef_NHV_Chg[40] := FALSE;
   UV_Bef_NHV_Chg[41] := FALSE;
   UV_Bef_NHV_Chg[42] := FALSE;
   UV_Bef_NHV_Chg[43] := FALSE;
   UV_Bef_NHV_Chg[44] := FALSE;
   UV_Bef_NHV_Chg[45] := FALSE;
   UV_Bef_NHV_Chg[46] := FALSE;
   UV_Bef_NHV_Chg[47] := FALSE;
   UV_Bef_NHV_Chg[48] := FALSE;
   UV_Bef_NHV_Chg[49] := FALSE;
   UV_Bef_NHV_Chg[50] := FALSE;
   UV_Bef_NHV_Chg[51] := FALSE;
   UV_Bef_NHV_Chg[52] := FALSE;
   UV_Bef_NHV_Chg[53] := FALSE;
   UV_Bef_NHV_Chg[54] := FALSE;
   UV_Bef_NHV_Chg[55] := FALSE;
   UV_Bef_NHV_Chg[56] := FALSE;
   UV_Bef_NHV_Chg[57] := FALSE;
   UV_Bef_NHV_Chg[58] := FALSE;
   UV_Bef_NHV_Chg[59] := FALSE;
   UV_Bef_NHV_Chg[60] := FALSE;
   UV_Bef_NHV_Chg[61] := FALSE;
   UV_Bef_NHV_Chg[62] := FALSE;
   UV_Bef_NHV_Chg[63] := FALSE;
   UV_Bef_NHV_Chg[64] := FALSE;
   UV_Bef_NHV_Chg[65] := FALSE;
   UV_Bef_NHV_Chg[66] := FALSE;
   UV_Bef_NHV_Chg[67] := FALSE;
   UV_Bef_NHV_Chg[68] := FALSE;
   UV_Bef_NHV_Chg[69] := FALSE;
   UV_Bef_NHV_Chg[70] := FALSE;
   UV_Bef_NHV_Chg[71] := FALSE;
   UV_Bef_NHV_Chg[72] := FALSE;
   UV_Bef_NHV_Chg[73] := FALSE;
   UV_Bef_NHV_Chg[74] := FALSE;
   UV_Bef_NHV_Chg[75] := FALSE;
   UV_Bef_NHV_Chg[76] := FALSE;
   UV_Bef_NHV_Chg[77] := FALSE;
   UV_Bef_NHV_Chg[78] := FALSE;
   UV_Bef_NHV_Chg[79] := FALSE;
   UV_Bef_NHV_Chg[80] := FALSE;
   UV_Bef_NHV_Chg[81] := FALSE;
   UV_Bef_NHV_Chg[82] := FALSE;
   UV_Bef_NHV_Chg[83] := FALSE;
   UV_Bef_NHV_Chg[84] := FALSE;
   UV_Bef_NHV_Chg[85] := FALSE;
   UV_Bef_NHV_Chg[86] := FALSE;
   UV_Bef_NHV_Chg[87] := FALSE;
   UV_Bef_NHV_Chg[88] := FALSE;
   UV_Bef_NHV_Chg[89] := FALSE;
   UV_Bef_NHV_Chg[90] := FALSE;
   UV_Bef_NHV_Chg[91] := FALSE;
   UV_Bef_NHV_Chg[92] := FALSE;
   UV_Bef_NHV_Chg[93] := FALSE;
   UV_Bef_NHV_Chg[94] := FALSE;
   UV_Bef_NHV_Chg[95] := FALSE;
   UV_Bef_NHV_Chg[96] := FALSE;
   UV_Bef_NHV_Chg[97] := FALSE;
   UV_Bef_NHV_Chg[98] := FALSE;
   UV_Bef_NHV_Chg[99] := FALSE;
   UV_Bef_NHV_Chg[100] := FALSE;
   UV_Bef_NHV_Chg[101] := FALSE;
   UV_Bef_NHV_Chg[102] := FALSE;
   UV_Bef_NHV_Chg[103] := FALSE;
   UV_Bef_NHV_Chg[104] := FALSE;
   UV_Bef_NHV_Chg[105] := FALSE;
   UV_Bef_NHV_Chg[106] := FALSE;
   UV_Bef_NHV_Chg[107] := FALSE;
   UV_Bef_NHV_Chg[108] := FALSE;
   UV_Bef_NHV_Chg[109] := FALSE;
   UV_Bef_NHV_Chg[110] := FALSE;
   UV_Bef_NHV_Chg[111] := FALSE;
   UV_Bef_NHV_Chg[112] := FALSE;
   UV_Bef_NHV_Chg[113] := FALSE;
   UV_Bef_NHV_Chg[114] := FALSE;
   UV_Bef_NHV_Chg[115] := FALSE;
   UV_Bef_NHV_Chg[116] := FALSE;
   UV_Bef_NHV_Chg[117] := FALSE;
   UV_Bef_NHV_Chg[118] := FALSE;
   UV_Bef_NHV_Chg[119] := FALSE;
   UV_Bef_NHV_Chg[120] := FALSE;
   UV_Bef_NHV_Chg[121] := FALSE;
   UV_Bef_NHV_Chg[122] := FALSE;
   UV_Bef_NHV_Chg[123] := FALSE;
   UV_Bef_NHV_Chg[124] := FALSE;
   UV_Bef_NHV_Chg[125] := FALSE;
   UV_Bef_NHV_Chg[126] := FALSE;
   UV_Bef_NHV_Chg[127] := FALSE;
   UV_Bef_NHV_Chg[128] := FALSE;
   UV_Bef_NHV_Chg[129] := FALSE;
   UV_Bef_NHV_Chg[130] := FALSE;
   UV_Bef_NHV_Chg[131] := FALSE;
   UV_Bef_NHV_Chg[132] := FALSE;
   UV_Bef_NHV_Chg[133] := FALSE;
   UV_Bef_NHV_Chg[134] := FALSE;
   UV_Bef_NHV_Chg[135] := FALSE;
   UV_Bef_NHV_Chg[136] := FALSE;
   UV_Bef_NHV_Chg[137] := FALSE;
   UV_Bef_NHV_Chg[138] := FALSE;
   UV_Bef_NHV_Chg[139] := FALSE;
   UV_Bef_NHV_Chg[140] := FALSE;
   UV_Bef_NHV_Chg[141] := FALSE;
   UV_Bef_NHV_Chg[142] := FALSE;
   UV_Bef_NHV_Chg[143] := FALSE;
   UV_Bef_NHV_Chg[144] := FALSE;
   UV_Meld_Chg[1] := TRUE;
   UV_Meld_Chg[2] := TRUE;
   UV_Meld_Chg[3] := TRUE;
   UV_Meld_Chg[4] := TRUE;
   UV_Meld_Chg[5] := TRUE;
   UV_Meld_Chg[6] := TRUE;
   UV_Meld_Chg[7] := TRUE;
   UV_Meld_Chg[8] := TRUE;
   UV_Meld_Chg[9] := TRUE;
   UV_Meld_Chg[10] := TRUE;
   UV_Meld_Chg[11] := TRUE;
   UV_Meld_Chg[12] := TRUE;
   UV_Meld_Chg[13] := TRUE;
   UV_Meld_Chg[14] := TRUE;
   UV_Meld_Chg[15] := TRUE;
   UV_Meld_Chg[16] := TRUE;
   UV_Meld_Chg[17] := TRUE;
   UV_Meld_Chg[18] := TRUE;
   UV_Meld_Chg[19] := TRUE;
   UV_Meld_Chg[20] := TRUE;
   UV_Meld_Chg[21] := TRUE;
   UV_Meld_Chg[22] := TRUE;
   UV_Meld_Chg[23] := FALSE;
   UV_Meld_Chg[24] := FALSE;
   UV_Meld_Chg[25] := FALSE;
   UV_Meld_Chg[26] := FALSE;
   UV_Meld_Chg[27] := FALSE;
   UV_Meld_Chg[28] := FALSE;
   UV_Meld_Chg[29] := FALSE;
   UV_Meld_Chg[30] := FALSE;
   UV_Meld_Chg[31] := FALSE;
   UV_Meld_Chg[32] := FALSE;
   UV_Meld_Chg[33] := FALSE;
   UV_Meld_Chg[34] := FALSE;
   UV_Meld_Chg[35] := FALSE;
   UV_Meld_Chg[36] := FALSE;
   UV_Meld_Chg[37] := FALSE;
   UV_Meld_Chg[38] := FALSE;
   UV_Meld_Chg[39] := FALSE;
   UV_Meld_Chg[40] := FALSE;
   UV_Meld_Chg[41] := FALSE;
   UV_Meld_Chg[42] := FALSE;
   UV_Meld_Chg[43] := FALSE;
   UV_Meld_Chg[44] := FALSE;
   UV_Meld_Chg[45] := FALSE;
   UV_Meld_Chg[46] := FALSE;
   UV_Meld_Chg[47] := FALSE;
   UV_Meld_Chg[48] := FALSE;
   UV_Meld_Chg[49] := FALSE;
   UV_Meld_Chg[50] := FALSE;
   UV_Meld_Chg[51] := FALSE;
   UV_Meld_Chg[52] := FALSE;
   UV_Meld_Chg[53] := FALSE;
   UV_Meld_Chg[54] := FALSE;
   UV_Meld_Chg[55] := FALSE;
   UV_Meld_Chg[56] := FALSE;
   UV_Meld_Chg[57] := FALSE;
   UV_Meld_Chg[58] := FALSE;
   UV_Meld_Chg[59] := FALSE;
   UV_Meld_Chg[60] := FALSE;
   UV_Meld_Chg[61] := FALSE;
   UV_Meld_Chg[62] := FALSE;
   UV_Meld_Chg[63] := FALSE;
   UV_Meld_Chg[64] := FALSE;
   UV_Meld_Chg[65] := FALSE;
   UV_Meld_Chg[66] := FALSE;
   UV_Meld_Chg[67] := FALSE;
   UV_Meld_Chg[68] := FALSE;
   UV_Meld_Chg[69] := FALSE;
   UV_Meld_Chg[70] := FALSE;
   UV_Meld_Chg[71] := FALSE;
   UV_Meld_Chg[72] := FALSE;
   UV_Meld_Chg[73] := FALSE;
   UV_Meld_Chg[74] := FALSE;
   UV_Meld_Chg[75] := FALSE;
   UV_Meld_Chg[76] := FALSE;
   UV_Meld_Chg[77] := FALSE;
   UV_Meld_Chg[78] := FALSE;
   UV_Meld_Chg[79] := FALSE;
   UV_Meld_Chg[80] := FALSE;
   UV_Meld_Chg[81] := FALSE;
   UV_Meld_Chg[82] := FALSE;
   UV_Meld_Chg[83] := FALSE;
   UV_Meld_Chg[84] := FALSE;
   UV_Meld_Chg[85] := FALSE;
   UV_Meld_Chg[86] := FALSE;
   UV_Meld_Chg[87] := FALSE;
   UV_Meld_Chg[88] := FALSE;
   UV_Meld_Chg[89] := FALSE;
   UV_Meld_Chg[90] := FALSE;
   UV_Meld_Chg[91] := FALSE;
   UV_Meld_Chg[92] := FALSE;
   UV_Meld_Chg[93] := FALSE;
   UV_Meld_Chg[94] := FALSE;
   UV_Meld_Chg[95] := FALSE;
   UV_Meld_Chg[96] := FALSE;
   UV_Meld_Chg[97] := FALSE;
   UV_Meld_Chg[98] := FALSE;
   UV_Meld_Chg[99] := FALSE;
   UV_Meld_Chg[100] := FALSE;
   UV_Meld_Chg[101] := FALSE;
   UV_Meld_Chg[102] := FALSE;
   UV_Meld_Chg[103] := FALSE;
   UV_Meld_Chg[104] := FALSE;
   UV_Meld_Chg[105] := FALSE;
   UV_Meld_Chg[106] := FALSE;
   UV_Meld_Chg[107] := FALSE;
   UV_Meld_Chg[108] := FALSE;
   UV_Meld_Chg[109] := FALSE;
   UV_Meld_Chg[110] := FALSE;
   UV_Meld_Chg[111] := FALSE;
   UV_Meld_Chg[112] := FALSE;
   UV_Meld_Chg[113] := FALSE;
   UV_Meld_Chg[114] := FALSE;
   UV_Meld_Chg[115] := FALSE;
   UV_Meld_Chg[116] := FALSE;
   UV_Meld_Chg[117] := FALSE;
   UV_Meld_Chg[118] := FALSE;
   UV_Meld_Chg[119] := FALSE;
   UV_Meld_Chg[120] := FALSE;
   UV_Meld_Chg[121] := FALSE;
   UV_Meld_Chg[122] := FALSE;
   UV_Meld_Chg[123] := FALSE;
   UV_Meld_Chg[124] := FALSE;
   UV_Meld_Chg[125] := FALSE;
   UV_Meld_Chg[126] := FALSE;
   UV_Meld_Chg[127] := FALSE;
   UV_Meld_Chg[128] := FALSE;
   UV_Meld_Chg[129] := FALSE;
   UV_Meld_Chg[130] := FALSE;
   UV_Meld_Chg[131] := FALSE;
   UV_Meld_Chg[132] := FALSE;
   UV_Meld_Chg[133] := FALSE;
   UV_Meld_Chg[134] := FALSE;
   UV_Meld_Chg[135] := FALSE;
   UV_Meld_Chg[136] := FALSE;
   UV_Meld_Chg[137] := FALSE;
   UV_Meld_Chg[138] := FALSE;
   UV_Meld_Chg[139] := FALSE;
   UV_Meld_Chg[140] := FALSE;
   UV_Meld_Chg[141] := FALSE;
   UV_Meld_Chg[142] := FALSE;
   UV_Meld_Chg[143] := FALSE;
   UV_Meld_Chg[144] := FALSE;
   UV_Prm_Chg[1] := FALSE;
   UV_Prm_Chg[2] := FALSE;
   UV_Prm_Chg[3] := FALSE;
   UV_Prm_Chg[4] := FALSE;
   UV_Prm_Chg[5] := FALSE;
   UV_Prm_Chg[6] := FALSE;
   UV_Prm_Chg[7] := FALSE;
   UV_Prm_Chg[8] := FALSE;
   UV_Prm_Chg[9] := FALSE;
   UV_Prm_Chg[10] := FALSE;
   UV_Prm_Chg[11] := FALSE;
   UV_Prm_Chg[12] := FALSE;
   UV_Prm_Chg[13] := FALSE;
   UV_Prm_Chg[14] := FALSE;
   UV_Prm_Chg[15] := FALSE;
   UV_Prm_Chg[16] := FALSE;
   UV_Prm_Chg[17] := FALSE;
   UV_Prm_Chg[18] := FALSE;
   UV_Prm_Chg[19] := FALSE;
   UV_Prm_Chg[20] := FALSE;
   UV_Prm_Chg[21] := FALSE;
   UV_Prm_Chg[22] := FALSE;
   UV_Prm_Chg[23] := FALSE;
   UV_Prm_Chg[24] := FALSE;
   UV_Prm_Chg[25] := FALSE;
   UV_Prm_Chg[26] := FALSE;
   UV_Prm_Chg[27] := FALSE;
   UV_Prm_Chg[28] := FALSE;
   UV_Prm_Chg[29] := FALSE;
   UV_Prm_Chg[30] := FALSE;
   UV_Prm_Chg[31] := FALSE;
   UV_Prm_Chg[32] := FALSE;
   UV_Prm_Chg[33] := FALSE;
   UV_Prm_Chg[34] := FALSE;
   UV_Prm_Chg[35] := FALSE;
   UV_Prm_Chg[36] := FALSE;
   UV_Prm_Chg[37] := FALSE;
   UV_Prm_Chg[38] := FALSE;
   UV_Prm_Chg[39] := FALSE;
   UV_Prm_Chg[40] := FALSE;
   UV_Prm_Chg[41] := FALSE;
   UV_Prm_Chg[42] := FALSE;
   UV_Prm_Chg[43] := FALSE;
   UV_Prm_Chg[44] := FALSE;
   UV_Prm_Chg[45] := FALSE;
   UV_Prm_Chg[46] := FALSE;
   UV_Prm_Chg[47] := FALSE;
   UV_Prm_Chg[48] := FALSE;
   UV_Prm_Chg[49] := FALSE;
   UV_Prm_Chg[50] := FALSE;
   UV_Prm_Chg[51] := FALSE;
   UV_Prm_Chg[52] := FALSE;
   UV_Prm_Chg[53] := FALSE;
   UV_Prm_Chg[54] := FALSE;
   UV_Prm_Chg[55] := FALSE;
   UV_Prm_Chg[56] := FALSE;
   UV_Prm_Chg[57] := FALSE;
   UV_Prm_Chg[58] := FALSE;
   UV_Prm_Chg[59] := FALSE;
   UV_Prm_Chg[60] := FALSE;
   UV_Prm_Chg[61] := FALSE;
   UV_Prm_Chg[62] := FALSE;
   UV_Prm_Chg[63] := FALSE;
   UV_Prm_Chg[64] := FALSE;
   UV_Prm_Chg[65] := FALSE;
   UV_Prm_Chg[66] := FALSE;
   UV_Prm_Chg[67] := FALSE;
   UV_Prm_Chg[68] := FALSE;
   UV_Prm_Chg[69] := FALSE;
   UV_Prm_Chg[70] := FALSE;
   UV_Prm_Chg[71] := FALSE;
   UV_Prm_Chg[72] := FALSE;
   UV_Prm_Chg[73] := FALSE;
   UV_Prm_Chg[74] := FALSE;
   UV_Prm_Chg[75] := FALSE;
   UV_Prm_Chg[76] := FALSE;
   UV_Prm_Chg[77] := FALSE;
   UV_Prm_Chg[78] := FALSE;
   UV_Prm_Chg[79] := FALSE;
   UV_Prm_Chg[80] := FALSE;
   UV_Prm_Chg[81] := FALSE;
   UV_Prm_Chg[82] := FALSE;
   UV_Prm_Chg[83] := FALSE;
   UV_Prm_Chg[84] := FALSE;
   UV_Prm_Chg[85] := FALSE;
   UV_Prm_Chg[86] := FALSE;
   UV_Prm_Chg[87] := FALSE;
   UV_Prm_Chg[88] := FALSE;
   UV_Prm_Chg[89] := FALSE;
   UV_Prm_Chg[90] := FALSE;
   UV_Prm_Chg[91] := FALSE;
   UV_Prm_Chg[92] := FALSE;
   UV_Prm_Chg[93] := FALSE;
   UV_Prm_Chg[94] := FALSE;
   UV_Prm_Chg[95] := FALSE;
   UV_Prm_Chg[96] := FALSE;
   UV_Prm_Chg[97] := FALSE;
   UV_Prm_Chg[98] := FALSE;
   UV_Prm_Chg[99] := FALSE;
   UV_Prm_Chg[100] := FALSE;
   UV_Prm_Chg[101] := FALSE;
   UV_Prm_Chg[102] := FALSE;
   UV_Prm_Chg[103] := FALSE;
   UV_Prm_Chg[104] := FALSE;
   UV_Prm_Chg[105] := FALSE;
   UV_Prm_Chg[106] := FALSE;
   UV_Prm_Chg[107] := FALSE;
   UV_Prm_Chg[108] := FALSE;
   UV_Prm_Chg[109] := FALSE;
   UV_Prm_Chg[110] := FALSE;
   UV_Prm_Chg[111] := FALSE;
   UV_Prm_Chg[112] := FALSE;
   UV_Prm_Chg[113] := FALSE;
   UV_Prm_Chg[114] := FALSE;
   UV_Prm_Chg[115] := FALSE;
   UV_Prm_Chg[116] := FALSE;
   UV_Prm_Chg[117] := FALSE;
   UV_Prm_Chg[118] := FALSE;
   UV_Prm_Chg[119] := FALSE;
   UV_Prm_Chg[120] := FALSE;
   UV_Prm_Chg[121] := FALSE;
   UV_Prm_Chg[122] := FALSE;
   UV_Prm_Chg[123] := FALSE;
   UV_Prm_Chg[124] := FALSE;
   UV_Prm_Chg[125] := FALSE;
   UV_Prm_Chg[126] := FALSE;
   UV_Prm_Chg[127] := FALSE;
   UV_Prm_Chg[128] := FALSE;
   UV_Prm_Chg[129] := FALSE;
   UV_Prm_Chg[130] := FALSE;
   UV_Prm_Chg[131] := FALSE;
   UV_Prm_Chg[132] := FALSE;
   UV_Prm_Chg[133] := FALSE;
   UV_Prm_Chg[134] := FALSE;
   UV_Prm_Chg[135] := FALSE;
   UV_Prm_Chg[136] := FALSE;
   UV_Prm_Chg[137] := FALSE;
   UV_Prm_Chg[138] := FALSE;
   UV_Prm_Chg[139] := FALSE;
   UV_Prm_Chg[140] := FALSE;
   UV_Prm_Chg[141] := FALSE;
   UV_Prm_Chg[142] := FALSE;
   UV_Prm_Chg[143] := FALSE;
   UV_Prm_Chg[144] := FALSE;

END_DATA_BLOCK

